SUBAPPLICATION Uebung_121 (* Übung zu ISOBUS Name *)
  (* Standard: 61499-2; Description: Copyright (c) 2025 Meisterschulen am Ostbahnhof This program and the accompanying materials are made available under the terms of the Eclipse Public License 2.0 which is available at https://www.eclipse.org/legal/epl-2.0/ SPDX-License-Identifier: EPL-2.0 *)
  (* Version 1.0, 2023-10-23, Franz Höpfinger, Meisterschulen am Ostbahnhof *)
  PACKAGE Uebungen;
  IMPORT isobus::pgn::ISOUSERHOME_e::thisMember;
  IMPORT isobus::pgn::ISO_CAN_NODE::NODE1;
  IMPORT Uebungen::const::Uebung_120_129::Filter::FLT_ALL_PASS;
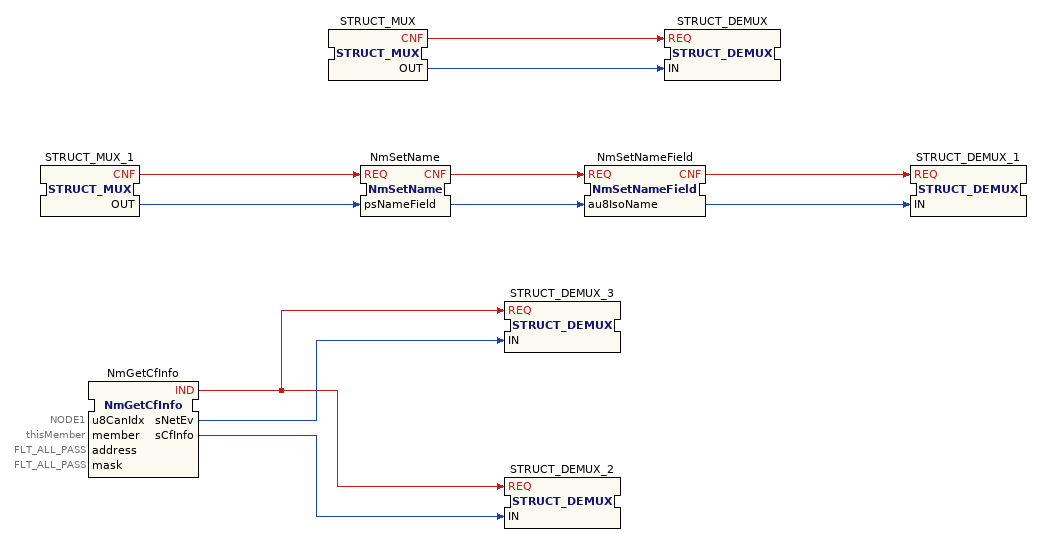
  FBS
    STRUCT_DEMUX : eclipse4diac::convert::STRUCT_DEMUX; {SET_ATTRIBUTE(StructuredType, isobus::pgn::NAMEFIELD_T)}
    STRUCT_MUX : eclipse4diac::convert::STRUCT_MUX; {SET_ATTRIBUTE(StructuredType, isobus::pgn::NAMEFIELD_T)}
    NmSetName : isobus::pgn::NmSetName;
    NmSetNameField : isobus::pgn::NmSetNameField;
    STRUCT_MUX_1 : eclipse4diac::convert::STRUCT_MUX; {SET_ATTRIBUTE(StructuredType, isobus::pgn::NAMEFIELD_T)}
    STRUCT_DEMUX_1 : eclipse4diac::convert::STRUCT_DEMUX; {SET_ATTRIBUTE(StructuredType, isobus::pgn::NAMEFIELD_T)}
    NmGetCfInfo : isobus::pgn::NmGetCfInfo(u8CanIdx := NODE1, member := thisMember, address := FLT_ALL_PASS, mask := FLT_ALL_PASS);
    STRUCT_DEMUX_2 : eclipse4diac::convert::STRUCT_DEMUX; {SET_ATTRIBUTE(StructuredType, isobus::pgn::CF_INFO_T)}
    STRUCT_DEMUX_3 : eclipse4diac::convert::STRUCT_DEMUX; {SET_ATTRIBUTE(StructuredType, isobus::pgn::ISONETEVENT_T)}
  END_FBS
  EVENT_CONNECTIONS
    STRUCT_MUX.CNF TO STRUCT_DEMUX.REQ;
    NmSetName.CNF TO NmSetNameField.REQ;
    STRUCT_MUX_1.CNF TO NmSetName.REQ;
    NmSetNameField.CNF TO STRUCT_DEMUX_1.REQ;
    NmGetCfInfo.IND TO STRUCT_DEMUX_3.REQ;
    NmGetCfInfo.IND TO STRUCT_DEMUX_2.REQ;
  END_CONNECTIONS
  DATA_CONNECTIONS
    STRUCT_MUX.OUT TO STRUCT_DEMUX.IN;
    STRUCT_MUX_1.OUT TO NmSetName.psNameField;
    NmSetName. TO NmSetNameField.au8IsoName;
    NmSetNameField. TO STRUCT_DEMUX_1.IN;
    NmGetCfInfo.sNetEv TO STRUCT_DEMUX_3.IN;
    NmGetCfInfo.sCfInfo TO STRUCT_DEMUX_2.IN;
  END_CONNECTIONS
END_SUBAPPLICATION
